TYPE CM_Vision_UDT :
STRUCT
	Input : DINT;
	
	PO_PV : DINT;
END_STRUCT
END_TYPE

(* stored: Version 1.1.0.1, ProductVersion 3.1.4024.13
   DUT CM_Vision_UDT: Id {2f9f2898-77d2-41aa-9383-0ef02fbf4b89} *)
